FUNCTION f_Setbit64 : LWORD
VAR_INPUT
  inVal   : LWORD;
  bitNo   : INT;
END_VAR
VAR
  wConst  : LWORD := 1;
END_VAR

f_Setbit64 := inVal OR SHL( wConst,INT_TO_SINT(bitNo) MOD 64 );

END_FUNCTION

(* stored: Version 1.1.0.1, ProductVersion 3.1.4022.18
   POU f_Setbit64: Id {3bde0ab1-c1b5-4ae3-8f39-8ea86e049c15}, SpecialFunc None *)
